{attribute 'qualified_only'}
{attribute 'strict'}
TYPE eTcoTaskTests :
(
	CallTasksBodiesOnly	:= 100,
	RestoreTasks,
    TaskInvokeAndWaitForDone := 300,
    TaskInvokeAfterDoneWithNoEmptyCycles,
    TaskInvokeAfterDoneWithOneEmptyCycle,
    TaskInvokeAfterDoneWithAbortCall,
    TaskInvokeAfterDoneWithRestoreCall,
    TaskAbortDuringExecutionAndInvoke,
    TaskError := 310,
    TaskInvokeAfterErrorNoRestoreNoEmptyCycles,
    TaskInvokeAfterErrorNoRestoreOneEmptyCycle,
    TaskInvokeAfterErrorWithRestore,
    TaskAbortDuringExecution,
    TaskMessage,
    IdentitiesTest,
    CheckAutoRestoreProperties,
    AutoRestoreOnStateChange,
    InvokeDisabledTask:=320,
    DisableExecutingTask,
    InvokeTaskThenDisable,
    DisableTaskInErrorStateEnableAndTriggerAgain,
    ElapsedTypeMeasurement:=330,
	TaskExecutingWithDoneAndErrorStatement := 340,
	TaskExecutingWithErrorAndDoneStatement
	
);
END_TYPE

(* stored: Version 1.1.0.1
   DUT eTcoTaskTests: Id {f67fe522-53fe-0e0a-32b0-2b622a8ec704} *)
